Fanuc TP program (LS listing): rsr0001.ls

/PROG  RSR0001
/ATTR
OWNER		= MNEDITOR;
COMMENT		= "";
PROG_SIZE	= 195;
CREATE		= DATE 26-07-24  TIME 22:53:36;
MODIFIED	= DATE 26-07-24  TIME 22:53:44;
FILE_NAME	= ;
VERSION		= 0;
LINE_COUNT	= 2;
MEMORY_SIZE	= 567;
PROTECT		= READ_WRITE;
TCD:  STACK_SIZE	= 0,
      TASK_PRIORITY	= 50,
      TIME_SLICE	= 0,
      BUSY_LAMP_OFF	= 0,
      ABORT_REQUEST	= 0,
      PAUSE_REQUEST	= 0;
DEFAULT_GROUP	= 1,*,*,*,*;
CONTROL_CODE	= 00000000 00000000;
LOCAL_REGISTERS	= 0,0,0;
/APPL

AUTO_SINGULARITY_HEADER;
  ENABLE_SINGULARITY_AVOIDANCE   : FALSE;
/MN
   1:  DO[112:ON :Power Cycled]=OFF ;
   2:  CALL __MAIN    ;
/POS
/END
